// TIA Portal V17 export
// export: Created 2025-06-20T10:18:09.7290963Z, ExportSetting WithDefaults, DisplayName Totally Integrated Automation Portal, DisplayVersion V17 Update 8, DisplayName TIA Portal Openness, DisplayVersion V17 Update 8, DisplayName TIA Portal Version Control Interface, DisplayVersion V17, DisplayName SINAMICS Startdrive Advanced, DisplayVersion V17 SP2, DisplayName SINAMICS Startdrive G110M, G120, G120C, G120D, G120P, G115D, DisplayVersion V17 SP2, DisplayName SINAMICS Startdrive G130, G150, S120, S150, SINAMICS MV, S210, DisplayVersion V17 SP2, DisplayName STEP 7 Professional, DisplayVersion V17 Update 8, DisplayName SINUMERIK ONE STEP 7 Toolbox, DisplayVersion V17 Update 12, DisplayName SINUMERIK ONE PLC Basic Program Plus, DisplayVersion V17 Update 12, DisplayName SINUMERIK 840D sl STEP 7 Toolbox, DisplayVersion V17 Update 12, DisplayName STEP 7 Safety, DisplayVersion V17 Update 6, DisplayName WinCC Advanced, DisplayVersion V17 Update 8
FUNCTION "FC370_NCK_M_CH8_UNIT_03" : Void   // FC370, LAD
TITLE = Channel 1 data
{ S7_Optimized_Access := 'FALSE' }
AUTHOR : ETXETAR
VERSION : 1.0
// stored: AutoNumber false, IsIECCheckEnabled false, SetENOAutomatically false, UDAEnableTagReadback false
BEGIN

REGION Network 1: ACKNOWLEDGE M704-FIXTURE 4 VERIFY PART AND TOOL IS CLAMPED DURING MACHINING (WHEN TRUE DO). TOGGLED / ACKNOWLEDGE M46-VERIFY FIXTURE 1 PART AND TOOL IS CLAMPED DURING
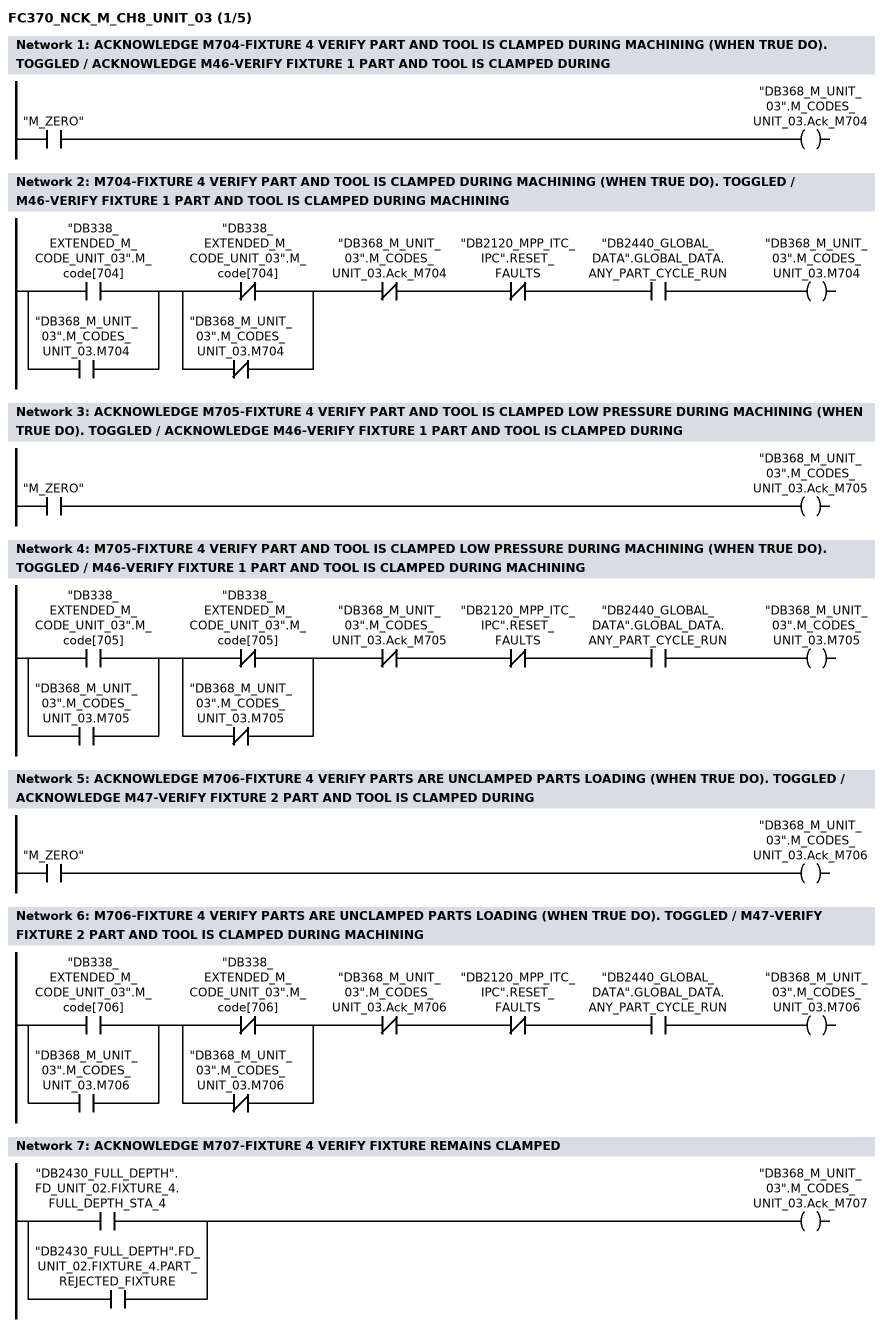
   RUNG wire#powerrail
      Contact( "M_ZERO" )
      Coil( "DB368_M_UNIT_03".M_CODES_UNIT_03.Ack_M704 )
   END_RUNG
   // the same network as SCL:
   "DB368_M_UNIT_03".M_CODES_UNIT_03.Ack_M704 := "M_ZERO";
END_REGION

REGION Network 2: M704-FIXTURE 4 VERIFY PART AND TOOL IS CLAMPED DURING MACHINING (WHEN TRUE DO). TOGGLED / M46-VERIFY FIXTURE 1 PART AND TOOL IS CLAMPED DURING MACHINING
   RUNG wire#powerrail
      Contact( "DB338_EXTENDED_M_CODE_UNIT_03".M_code[704] )
      wire#w1
      I_Contact( "DB338_EXTENDED_M_CODE_UNIT_03".M_code[704] )
      wire#w2
      I_Contact( "DB368_M_UNIT_03".M_CODES_UNIT_03.Ack_M704 )
      I_Contact( "DB2120_MPP_ITC_IPC".RESET_FAULTS )
      Contact( "DB2440_GLOBAL_DATA".GLOBAL_DATA.ANY_PART_CYCLE_RUN )
      Coil( "DB368_M_UNIT_03".M_CODES_UNIT_03.M704 )
   END_RUNG
   RUNG wire#powerrail
      Contact( "DB368_M_UNIT_03".M_CODES_UNIT_03.M704 )
   END_RUNG wire#w1
   RUNG wire#w1
      I_Contact( "DB368_M_UNIT_03".M_CODES_UNIT_03.M704 )
   END_RUNG wire#w2
   // the same network as SCL:
   "DB368_M_UNIT_03".M_CODES_UNIT_03.M704 := ("DB338_EXTENDED_M_CODE_UNIT_03".M_code[704] OR "DB368_M_UNIT_03".M_CODES_UNIT_03.M704) AND (NOT "DB338_EXTENDED_M_CODE_UNIT_03".M_code[704] OR NOT "DB368_M_UNIT_03".M_CODES_UNIT_03.M704) AND NOT "DB368_M_UNIT_03".M_CODES_UNIT_03.Ack_M704 AND NOT "DB2120_MPP_ITC_IPC".RESET_FAULTS AND "DB2440_GLOBAL_DATA".GLOBAL_DATA.ANY_PART_CYCLE_RUN;
END_REGION

REGION Network 3: ACKNOWLEDGE M705-FIXTURE 4 VERIFY PART AND TOOL IS CLAMPED LOW PRESSURE DURING MACHINING (WHEN TRUE DO). TOGGLED / ACKNOWLEDGE M46-VERIFY FIXTURE 1 PART AND TOOL IS CLAMPED DURING
   RUNG wire#powerrail
      Contact( "M_ZERO" )
      Coil( "DB368_M_UNIT_03".M_CODES_UNIT_03.Ack_M705 )
   END_RUNG
   // the same network as SCL:
   "DB368_M_UNIT_03".M_CODES_UNIT_03.Ack_M705 := "M_ZERO";
END_REGION

REGION Network 4: M705-FIXTURE 4 VERIFY PART AND TOOL IS CLAMPED LOW PRESSURE DURING MACHINING (WHEN TRUE DO). TOGGLED / M46-VERIFY FIXTURE 1 PART AND TOOL IS CLAMPED DURING MACHINING
   RUNG wire#powerrail
      Contact( "DB338_EXTENDED_M_CODE_UNIT_03".M_code[705] )
      wire#w1
      I_Contact( "DB338_EXTENDED_M_CODE_UNIT_03".M_code[705] )
      wire#w2
      I_Contact( "DB368_M_UNIT_03".M_CODES_UNIT_03.Ack_M705 )
      I_Contact( "DB2120_MPP_ITC_IPC".RESET_FAULTS )
      Contact( "DB2440_GLOBAL_DATA".GLOBAL_DATA.ANY_PART_CYCLE_RUN )
      Coil( "DB368_M_UNIT_03".M_CODES_UNIT_03.M705 )
   END_RUNG
   RUNG wire#powerrail
      Contact( "DB368_M_UNIT_03".M_CODES_UNIT_03.M705 )
   END_RUNG wire#w1
   RUNG wire#w1
      I_Contact( "DB368_M_UNIT_03".M_CODES_UNIT_03.M705 )
   END_RUNG wire#w2
   // the same network as SCL:
   "DB368_M_UNIT_03".M_CODES_UNIT_03.M705 := ("DB338_EXTENDED_M_CODE_UNIT_03".M_code[705] OR "DB368_M_UNIT_03".M_CODES_UNIT_03.M705) AND (NOT "DB338_EXTENDED_M_CODE_UNIT_03".M_code[705] OR NOT "DB368_M_UNIT_03".M_CODES_UNIT_03.M705) AND NOT "DB368_M_UNIT_03".M_CODES_UNIT_03.Ack_M705 AND NOT "DB2120_MPP_ITC_IPC".RESET_FAULTS AND "DB2440_GLOBAL_DATA".GLOBAL_DATA.ANY_PART_CYCLE_RUN;
END_REGION

REGION Network 5: ACKNOWLEDGE M706-FIXTURE 4 VERIFY PARTS ARE UNCLAMPED PARTS LOADING (WHEN TRUE DO). TOGGLED / ACKNOWLEDGE M47-VERIFY FIXTURE 2 PART AND TOOL IS CLAMPED DURING
   RUNG wire#powerrail
      Contact( "M_ZERO" )
      Coil( "DB368_M_UNIT_03".M_CODES_UNIT_03.Ack_M706 )
   END_RUNG
   // the same network as SCL:
   "DB368_M_UNIT_03".M_CODES_UNIT_03.Ack_M706 := "M_ZERO";
END_REGION

REGION Network 6: M706-FIXTURE 4 VERIFY PARTS ARE UNCLAMPED PARTS LOADING (WHEN TRUE DO). TOGGLED / M47-VERIFY FIXTURE 2 PART AND TOOL IS CLAMPED DURING MACHINING
   RUNG wire#powerrail
      Contact( "DB338_EXTENDED_M_CODE_UNIT_03".M_code[706] )
      wire#w1
      I_Contact( "DB338_EXTENDED_M_CODE_UNIT_03".M_code[706] )
      wire#w2
      I_Contact( "DB368_M_UNIT_03".M_CODES_UNIT_03.Ack_M706 )
      I_Contact( "DB2120_MPP_ITC_IPC".RESET_FAULTS )
      Contact( "DB2440_GLOBAL_DATA".GLOBAL_DATA.ANY_PART_CYCLE_RUN )
      Coil( "DB368_M_UNIT_03".M_CODES_UNIT_03.M706 )
   END_RUNG
   RUNG wire#powerrail
      Contact( "DB368_M_UNIT_03".M_CODES_UNIT_03.M706 )
   END_RUNG wire#w1
   RUNG wire#w1
      I_Contact( "DB368_M_UNIT_03".M_CODES_UNIT_03.M706 )
   END_RUNG wire#w2
   // the same network as SCL:
   "DB368_M_UNIT_03".M_CODES_UNIT_03.M706 := ("DB338_EXTENDED_M_CODE_UNIT_03".M_code[706] OR "DB368_M_UNIT_03".M_CODES_UNIT_03.M706) AND (NOT "DB338_EXTENDED_M_CODE_UNIT_03".M_code[706] OR NOT "DB368_M_UNIT_03".M_CODES_UNIT_03.M706) AND NOT "DB368_M_UNIT_03".M_CODES_UNIT_03.Ack_M706 AND NOT "DB2120_MPP_ITC_IPC".RESET_FAULTS AND "DB2440_GLOBAL_DATA".GLOBAL_DATA.ANY_PART_CYCLE_RUN;
END_REGION

REGION Network 7: ACKNOWLEDGE M707-FIXTURE 4 VERIFY FIXTURE REMAINS CLAMPED
   RUNG wire#powerrail
      Contact( "DB2430_FULL_DEPTH".FD_UNIT_02.FIXTURE_4.FULL_DEPTH_STA_4 )
      wire#w1
      Coil( "DB368_M_UNIT_03".M_CODES_UNIT_03.Ack_M707 )
   END_RUNG
   RUNG wire#powerrail
      Contact( "DB2430_FULL_DEPTH".FD_UNIT_02.FIXTURE_4.PART_REJECTED_FIXTURE )
   END_RUNG wire#w1
   // the same network as SCL:
   "DB368_M_UNIT_03".M_CODES_UNIT_03.Ack_M707 := "DB2430_FULL_DEPTH".FD_UNIT_02.FIXTURE_4.FULL_DEPTH_STA_4 OR "DB2430_FULL_DEPTH".FD_UNIT_02.FIXTURE_4.PART_REJECTED_FIXTURE;
END_REGION

REGION Network 8: M707-FIXTURE 4 VERIFY FIXTURE REMAINS CLAMPED
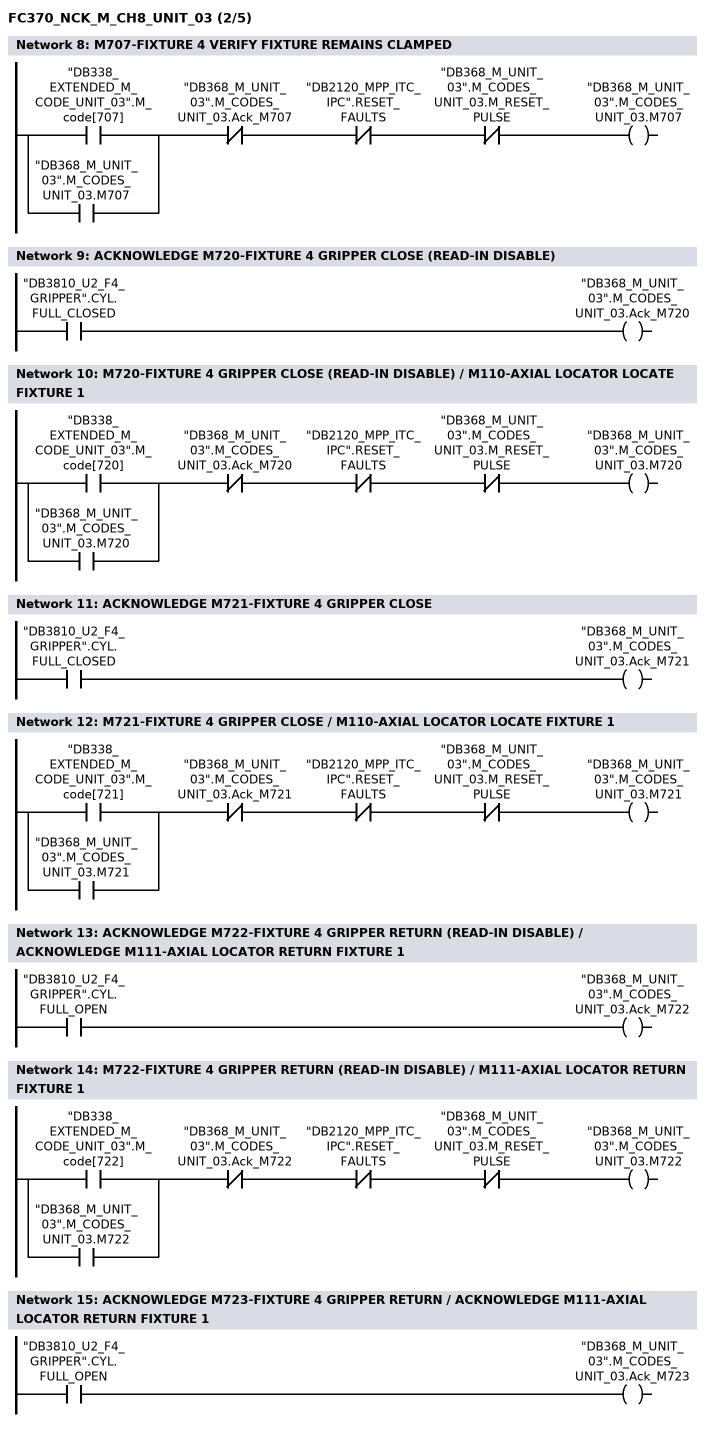
   RUNG wire#powerrail
      Contact( "DB338_EXTENDED_M_CODE_UNIT_03".M_code[707] )
      wire#w1
      I_Contact( "DB368_M_UNIT_03".M_CODES_UNIT_03.Ack_M707 )
      I_Contact( "DB2120_MPP_ITC_IPC".RESET_FAULTS )
      I_Contact( "DB368_M_UNIT_03".M_CODES_UNIT_03.M_RESET_PULSE )
      Coil( "DB368_M_UNIT_03".M_CODES_UNIT_03.M707 )
   END_RUNG
   RUNG wire#powerrail
      Contact( "DB368_M_UNIT_03".M_CODES_UNIT_03.M707 )
   END_RUNG wire#w1
   // the same network as SCL:
   "DB368_M_UNIT_03".M_CODES_UNIT_03.M707 := ("DB338_EXTENDED_M_CODE_UNIT_03".M_code[707] OR "DB368_M_UNIT_03".M_CODES_UNIT_03.M707) AND NOT "DB368_M_UNIT_03".M_CODES_UNIT_03.Ack_M707 AND NOT "DB2120_MPP_ITC_IPC".RESET_FAULTS AND NOT "DB368_M_UNIT_03".M_CODES_UNIT_03.M_RESET_PULSE;
END_REGION

REGION Network 9: ACKNOWLEDGE M720-FIXTURE 4 GRIPPER CLOSE (READ-IN DISABLE)
   RUNG wire#powerrail
      Contact( "DB3810_U2_F4_GRIPPER".CYL.FULL_CLOSED )
      Coil( "DB368_M_UNIT_03".M_CODES_UNIT_03.Ack_M720 )
   END_RUNG
   // the same network as SCL:
   "DB368_M_UNIT_03".M_CODES_UNIT_03.Ack_M720 := "DB3810_U2_F4_GRIPPER".CYL.FULL_CLOSED;
END_REGION

REGION Network 10: M720-FIXTURE 4 GRIPPER CLOSE (READ-IN DISABLE) / M110-AXIAL LOCATOR LOCATE FIXTURE 1
   RUNG wire#powerrail
      Contact( "DB338_EXTENDED_M_CODE_UNIT_03".M_code[720] )
      wire#w1
      I_Contact( "DB368_M_UNIT_03".M_CODES_UNIT_03.Ack_M720 )
      I_Contact( "DB2120_MPP_ITC_IPC".RESET_FAULTS )
      I_Contact( "DB368_M_UNIT_03".M_CODES_UNIT_03.M_RESET_PULSE )
      Coil( "DB368_M_UNIT_03".M_CODES_UNIT_03.M720 )
   END_RUNG
   RUNG wire#powerrail
      Contact( "DB368_M_UNIT_03".M_CODES_UNIT_03.M720 )
   END_RUNG wire#w1
   // the same network as SCL:
   "DB368_M_UNIT_03".M_CODES_UNIT_03.M720 := ("DB338_EXTENDED_M_CODE_UNIT_03".M_code[720] OR "DB368_M_UNIT_03".M_CODES_UNIT_03.M720) AND NOT "DB368_M_UNIT_03".M_CODES_UNIT_03.Ack_M720 AND NOT "DB2120_MPP_ITC_IPC".RESET_FAULTS AND NOT "DB368_M_UNIT_03".M_CODES_UNIT_03.M_RESET_PULSE;
END_REGION

REGION Network 11: ACKNOWLEDGE M721-FIXTURE 4 GRIPPER CLOSE
   RUNG wire#powerrail
      Contact( "DB3810_U2_F4_GRIPPER".CYL.FULL_CLOSED )
      Coil( "DB368_M_UNIT_03".M_CODES_UNIT_03.Ack_M721 )
   END_RUNG
   // the same network as SCL:
   "DB368_M_UNIT_03".M_CODES_UNIT_03.Ack_M721 := "DB3810_U2_F4_GRIPPER".CYL.FULL_CLOSED;
END_REGION

REGION Network 12: M721-FIXTURE 4 GRIPPER CLOSE / M110-AXIAL LOCATOR LOCATE FIXTURE 1
   RUNG wire#powerrail
      Contact( "DB338_EXTENDED_M_CODE_UNIT_03".M_code[721] )
      wire#w1
      I_Contact( "DB368_M_UNIT_03".M_CODES_UNIT_03.Ack_M721 )
      I_Contact( "DB2120_MPP_ITC_IPC".RESET_FAULTS )
      I_Contact( "DB368_M_UNIT_03".M_CODES_UNIT_03.M_RESET_PULSE )
      Coil( "DB368_M_UNIT_03".M_CODES_UNIT_03.M721 )
   END_RUNG
   RUNG wire#powerrail
      Contact( "DB368_M_UNIT_03".M_CODES_UNIT_03.M721 )
   END_RUNG wire#w1
   // the same network as SCL:
   "DB368_M_UNIT_03".M_CODES_UNIT_03.M721 := ("DB338_EXTENDED_M_CODE_UNIT_03".M_code[721] OR "DB368_M_UNIT_03".M_CODES_UNIT_03.M721) AND NOT "DB368_M_UNIT_03".M_CODES_UNIT_03.Ack_M721 AND NOT "DB2120_MPP_ITC_IPC".RESET_FAULTS AND NOT "DB368_M_UNIT_03".M_CODES_UNIT_03.M_RESET_PULSE;
END_REGION

REGION Network 13: ACKNOWLEDGE M722-FIXTURE 4 GRIPPER RETURN (READ-IN DISABLE) / ACKNOWLEDGE M111-AXIAL LOCATOR RETURN FIXTURE 1
   RUNG wire#powerrail
      Contact( "DB3810_U2_F4_GRIPPER".CYL.FULL_OPEN )
      Coil( "DB368_M_UNIT_03".M_CODES_UNIT_03.Ack_M722 )
   END_RUNG
   // the same network as SCL:
   "DB368_M_UNIT_03".M_CODES_UNIT_03.Ack_M722 := "DB3810_U2_F4_GRIPPER".CYL.FULL_OPEN;
END_REGION

REGION Network 14: M722-FIXTURE 4 GRIPPER RETURN (READ-IN DISABLE) / M111-AXIAL LOCATOR RETURN FIXTURE 1
   RUNG wire#powerrail
      Contact( "DB338_EXTENDED_M_CODE_UNIT_03".M_code[722] )
      wire#w1
      I_Contact( "DB368_M_UNIT_03".M_CODES_UNIT_03.Ack_M722 )
      I_Contact( "DB2120_MPP_ITC_IPC".RESET_FAULTS )
      I_Contact( "DB368_M_UNIT_03".M_CODES_UNIT_03.M_RESET_PULSE )
      Coil( "DB368_M_UNIT_03".M_CODES_UNIT_03.M722 )
   END_RUNG
   RUNG wire#powerrail
      Contact( "DB368_M_UNIT_03".M_CODES_UNIT_03.M722 )
   END_RUNG wire#w1
   // the same network as SCL:
   "DB368_M_UNIT_03".M_CODES_UNIT_03.M722 := ("DB338_EXTENDED_M_CODE_UNIT_03".M_code[722] OR "DB368_M_UNIT_03".M_CODES_UNIT_03.M722) AND NOT "DB368_M_UNIT_03".M_CODES_UNIT_03.Ack_M722 AND NOT "DB2120_MPP_ITC_IPC".RESET_FAULTS AND NOT "DB368_M_UNIT_03".M_CODES_UNIT_03.M_RESET_PULSE;
END_REGION

REGION Network 15: ACKNOWLEDGE M723-FIXTURE 4 GRIPPER RETURN / ACKNOWLEDGE M111-AXIAL LOCATOR RETURN FIXTURE 1
   RUNG wire#powerrail
      Contact( "DB3810_U2_F4_GRIPPER".CYL.FULL_OPEN )
      Coil( "DB368_M_UNIT_03".M_CODES_UNIT_03.Ack_M723 )
   END_RUNG
   // the same network as SCL:
   "DB368_M_UNIT_03".M_CODES_UNIT_03.Ack_M723 := "DB3810_U2_F4_GRIPPER".CYL.FULL_OPEN;
END_REGION

REGION Network 16: M723-FIXTURE 4 GRIPPER RETURN / M111-AXIAL LOCATOR RETURN FIXTURE 1
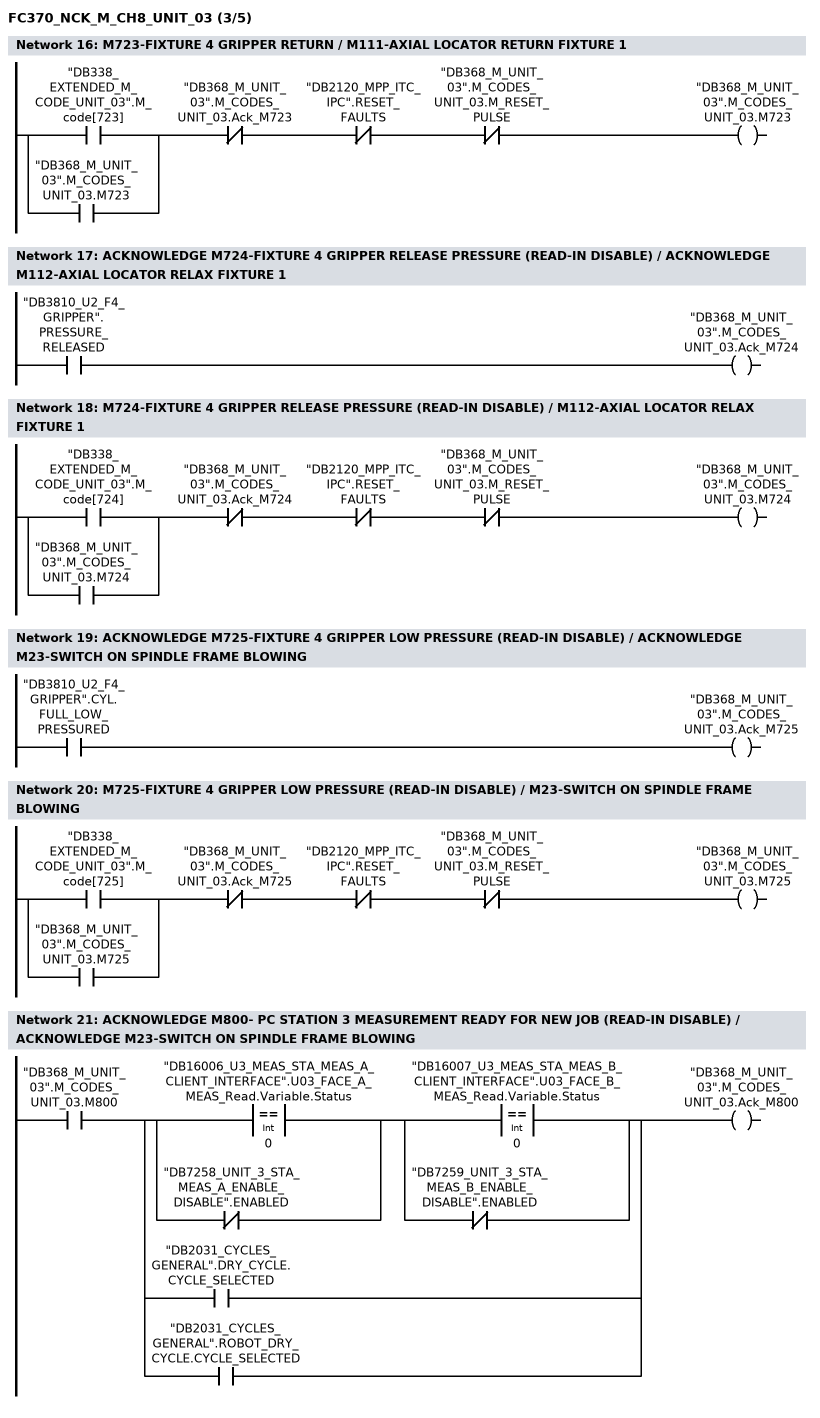
   RUNG wire#powerrail
      Contact( "DB338_EXTENDED_M_CODE_UNIT_03".M_code[723] )
      wire#w1
      I_Contact( "DB368_M_UNIT_03".M_CODES_UNIT_03.Ack_M723 )
      I_Contact( "DB2120_MPP_ITC_IPC".RESET_FAULTS )
      I_Contact( "DB368_M_UNIT_03".M_CODES_UNIT_03.M_RESET_PULSE )
      Coil( "DB368_M_UNIT_03".M_CODES_UNIT_03.M723 )
   END_RUNG
   RUNG wire#powerrail
      Contact( "DB368_M_UNIT_03".M_CODES_UNIT_03.M723 )
   END_RUNG wire#w1
   // the same network as SCL:
   "DB368_M_UNIT_03".M_CODES_UNIT_03.M723 := ("DB338_EXTENDED_M_CODE_UNIT_03".M_code[723] OR "DB368_M_UNIT_03".M_CODES_UNIT_03.M723) AND NOT "DB368_M_UNIT_03".M_CODES_UNIT_03.Ack_M723 AND NOT "DB2120_MPP_ITC_IPC".RESET_FAULTS AND NOT "DB368_M_UNIT_03".M_CODES_UNIT_03.M_RESET_PULSE;
END_REGION

REGION Network 17: ACKNOWLEDGE M724-FIXTURE 4 GRIPPER RELEASE PRESSURE (READ-IN DISABLE) / ACKNOWLEDGE M112-AXIAL LOCATOR RELAX FIXTURE 1
   RUNG wire#powerrail
      Contact( "DB3810_U2_F4_GRIPPER".PRESSURE_RELEASED )
      Coil( "DB368_M_UNIT_03".M_CODES_UNIT_03.Ack_M724 )
   END_RUNG
   // the same network as SCL:
   "DB368_M_UNIT_03".M_CODES_UNIT_03.Ack_M724 := "DB3810_U2_F4_GRIPPER".PRESSURE_RELEASED;
END_REGION

REGION Network 18: M724-FIXTURE 4 GRIPPER RELEASE PRESSURE (READ-IN DISABLE) / M112-AXIAL LOCATOR RELAX FIXTURE 1
   RUNG wire#powerrail
      Contact( "DB338_EXTENDED_M_CODE_UNIT_03".M_code[724] )
      wire#w1
      I_Contact( "DB368_M_UNIT_03".M_CODES_UNIT_03.Ack_M724 )
      I_Contact( "DB2120_MPP_ITC_IPC".RESET_FAULTS )
      I_Contact( "DB368_M_UNIT_03".M_CODES_UNIT_03.M_RESET_PULSE )
      Coil( "DB368_M_UNIT_03".M_CODES_UNIT_03.M724 )
   END_RUNG
   RUNG wire#powerrail
      Contact( "DB368_M_UNIT_03".M_CODES_UNIT_03.M724 )
   END_RUNG wire#w1
   // the same network as SCL:
   "DB368_M_UNIT_03".M_CODES_UNIT_03.M724 := ("DB338_EXTENDED_M_CODE_UNIT_03".M_code[724] OR "DB368_M_UNIT_03".M_CODES_UNIT_03.M724) AND NOT "DB368_M_UNIT_03".M_CODES_UNIT_03.Ack_M724 AND NOT "DB2120_MPP_ITC_IPC".RESET_FAULTS AND NOT "DB368_M_UNIT_03".M_CODES_UNIT_03.M_RESET_PULSE;
END_REGION

REGION Network 19: ACKNOWLEDGE M725-FIXTURE 4 GRIPPER LOW PRESSURE (READ-IN DISABLE) / ACKNOWLEDGE M23-SWITCH ON SPINDLE FRAME BLOWING
   RUNG wire#powerrail
      Contact( "DB3810_U2_F4_GRIPPER".CYL.FULL_LOW_PRESSURED )
      Coil( "DB368_M_UNIT_03".M_CODES_UNIT_03.Ack_M725 )
   END_RUNG
   // the same network as SCL:
   "DB368_M_UNIT_03".M_CODES_UNIT_03.Ack_M725 := "DB3810_U2_F4_GRIPPER".CYL.FULL_LOW_PRESSURED;
END_REGION

REGION Network 20: M725-FIXTURE 4 GRIPPER LOW PRESSURE (READ-IN DISABLE) / M23-SWITCH ON SPINDLE FRAME BLOWING
   RUNG wire#powerrail
      Contact( "DB338_EXTENDED_M_CODE_UNIT_03".M_code[725] )
      wire#w1
      I_Contact( "DB368_M_UNIT_03".M_CODES_UNIT_03.Ack_M725 )
      I_Contact( "DB2120_MPP_ITC_IPC".RESET_FAULTS )
      I_Contact( "DB368_M_UNIT_03".M_CODES_UNIT_03.M_RESET_PULSE )
      Coil( "DB368_M_UNIT_03".M_CODES_UNIT_03.M725 )
   END_RUNG
   RUNG wire#powerrail
      Contact( "DB368_M_UNIT_03".M_CODES_UNIT_03.M725 )
   END_RUNG wire#w1
   // the same network as SCL:
   "DB368_M_UNIT_03".M_CODES_UNIT_03.M725 := ("DB338_EXTENDED_M_CODE_UNIT_03".M_code[725] OR "DB368_M_UNIT_03".M_CODES_UNIT_03.M725) AND NOT "DB368_M_UNIT_03".M_CODES_UNIT_03.Ack_M725 AND NOT "DB2120_MPP_ITC_IPC".RESET_FAULTS AND NOT "DB368_M_UNIT_03".M_CODES_UNIT_03.M_RESET_PULSE;
END_REGION

REGION Network 21: ACKNOWLEDGE M800- PC STATION 3 MEASUREMENT READY FOR NEW JOB (READ-IN DISABLE) / ACKNOWLEDGE M23-SWITCH ON SPINDLE FRAME BLOWING
   RUNG wire#powerrail
      Contact( "DB368_M_UNIT_03".M_CODES_UNIT_03.M800 )
      wire#w1
      { S7_Templates := "SrcType := Int" } EQ_Contact(in1 := "DB16006_U3_MEAS_STA_MEAS_A_CLIENT_INTERFACE".U03_FACE_A_MEAS_Read.Variable.Status, in2 := 0)
      wire#w2
      { S7_Templates := "SrcType := Int" } EQ_Contact(in1 := "DB16007_U3_MEAS_STA_MEAS_B_CLIENT_INTERFACE".U03_FACE_B_MEAS_Read.Variable.Status, in2 := 0)
      wire#w3
      Coil( "DB368_M_UNIT_03".M_CODES_UNIT_03.Ack_M800 )
   END_RUNG
   RUNG wire#w1
      I_Contact( "DB7258_UNIT_3_STA_MEAS_A_ENABLE_DISABLE".ENABLED )
   END_RUNG wire#w2
   RUNG wire#w2
      I_Contact( "DB7259_UNIT_3_STA_MEAS_B_ENABLE_DISABLE".ENABLED )
   END_RUNG wire#w3
   RUNG wire#w1
      Contact( "DB2031_CYCLES_GENERAL".DRY_CYCLE.CYCLE_SELECTED )
   END_RUNG wire#w3
   RUNG wire#w1
      Contact( "DB2031_CYCLES_GENERAL".ROBOT_DRY_CYCLE.CYCLE_SELECTED )
   END_RUNG wire#w3
   // the same network as SCL:
   "DB368_M_UNIT_03".M_CODES_UNIT_03.Ack_M800 := "DB368_M_UNIT_03".M_CODES_UNIT_03.M800 AND (((("DB16006_U3_MEAS_STA_MEAS_A_CLIENT_INTERFACE".U03_FACE_A_MEAS_Read.Variable.Status = 0) OR NOT "DB7258_UNIT_3_STA_MEAS_A_ENABLE_DISABLE".ENABLED) AND (("DB16007_U3_MEAS_STA_MEAS_B_CLIENT_INTERFACE".U03_FACE_B_MEAS_Read.Variable.Status = 0) OR NOT "DB7259_UNIT_3_STA_MEAS_B_ENABLE_DISABLE".ENABLED)) OR "DB2031_CYCLES_GENERAL".DRY_CYCLE.CYCLE_SELECTED OR "DB2031_CYCLES_GENERAL".ROBOT_DRY_CYCLE.CYCLE_SELECTED);
END_REGION

REGION Network 22: M800- PC STATION 3 MEASUREMENT READY FOR NEW JOB (READ-IN DISABLE) / M23-SWITCH ON SPINDLE FRAME BLOWING
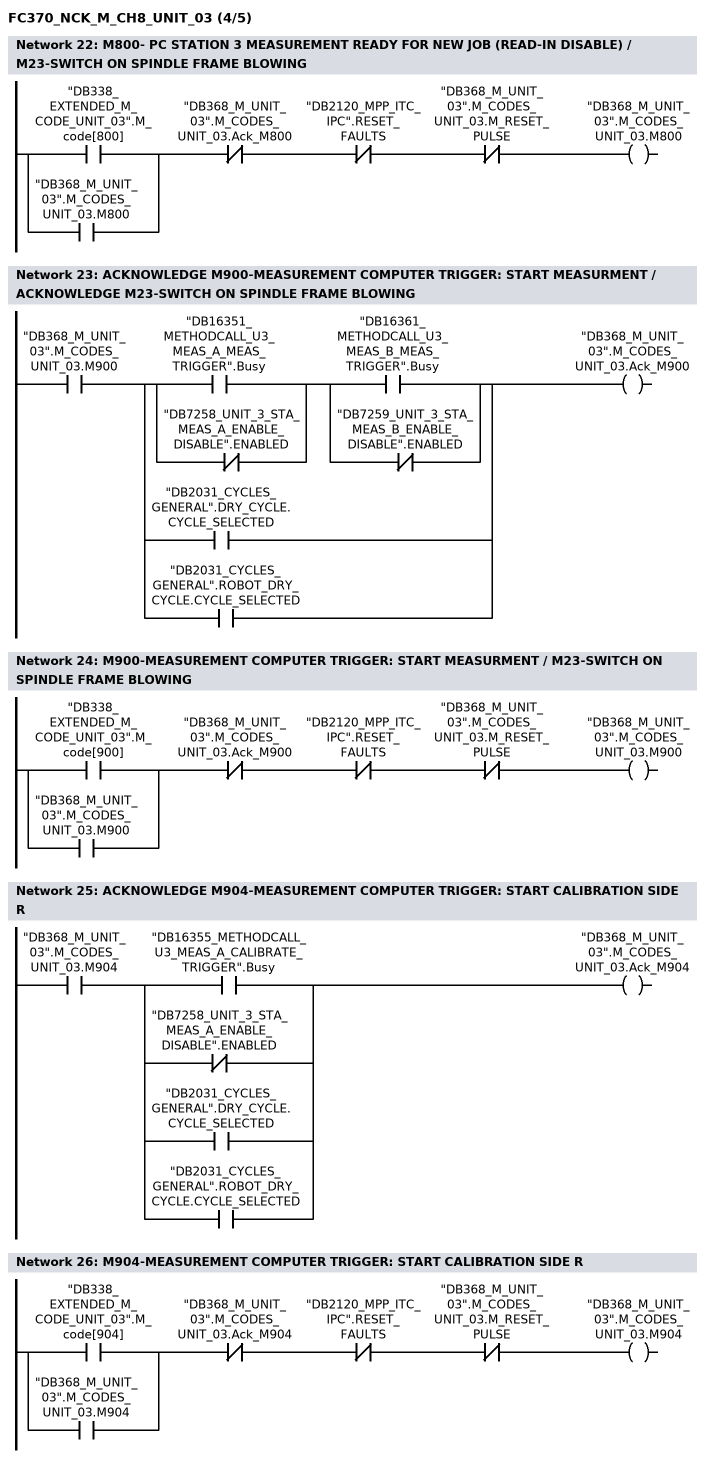
   RUNG wire#powerrail
      Contact( "DB338_EXTENDED_M_CODE_UNIT_03".M_code[800] )
      wire#w1
      I_Contact( "DB368_M_UNIT_03".M_CODES_UNIT_03.Ack_M800 )
      I_Contact( "DB2120_MPP_ITC_IPC".RESET_FAULTS )
      I_Contact( "DB368_M_UNIT_03".M_CODES_UNIT_03.M_RESET_PULSE )
      Coil( "DB368_M_UNIT_03".M_CODES_UNIT_03.M800 )
   END_RUNG
   RUNG wire#powerrail
      Contact( "DB368_M_UNIT_03".M_CODES_UNIT_03.M800 )
   END_RUNG wire#w1
   // the same network as SCL:
   "DB368_M_UNIT_03".M_CODES_UNIT_03.M800 := ("DB338_EXTENDED_M_CODE_UNIT_03".M_code[800] OR "DB368_M_UNIT_03".M_CODES_UNIT_03.M800) AND NOT "DB368_M_UNIT_03".M_CODES_UNIT_03.Ack_M800 AND NOT "DB2120_MPP_ITC_IPC".RESET_FAULTS AND NOT "DB368_M_UNIT_03".M_CODES_UNIT_03.M_RESET_PULSE;
END_REGION

REGION Network 23: ACKNOWLEDGE M900-MEASUREMENT COMPUTER TRIGGER: START MEASURMENT / ACKNOWLEDGE M23-SWITCH ON SPINDLE FRAME BLOWING
   RUNG wire#powerrail
      Contact( "DB368_M_UNIT_03".M_CODES_UNIT_03.M900 )
      wire#w1
      Contact( "DB16351_METHODCALL_U3_MEAS_A_MEAS_TRIGGER".Busy )
      wire#w2
      Contact( "DB16361_METHODCALL_U3_MEAS_B_MEAS_TRIGGER".Busy )
      wire#w3
      Coil( "DB368_M_UNIT_03".M_CODES_UNIT_03.Ack_M900 )
   END_RUNG
   RUNG wire#w1
      I_Contact( "DB7258_UNIT_3_STA_MEAS_A_ENABLE_DISABLE".ENABLED )
   END_RUNG wire#w2
   RUNG wire#w2
      I_Contact( "DB7259_UNIT_3_STA_MEAS_B_ENABLE_DISABLE".ENABLED )
   END_RUNG wire#w3
   RUNG wire#w1
      Contact( "DB2031_CYCLES_GENERAL".DRY_CYCLE.CYCLE_SELECTED )
   END_RUNG wire#w3
   RUNG wire#w1
      Contact( "DB2031_CYCLES_GENERAL".ROBOT_DRY_CYCLE.CYCLE_SELECTED )
   END_RUNG wire#w3
   // the same network as SCL:
   "DB368_M_UNIT_03".M_CODES_UNIT_03.Ack_M900 := "DB368_M_UNIT_03".M_CODES_UNIT_03.M900 AND ((("DB16351_METHODCALL_U3_MEAS_A_MEAS_TRIGGER".Busy OR NOT "DB7258_UNIT_3_STA_MEAS_A_ENABLE_DISABLE".ENABLED) AND ("DB16361_METHODCALL_U3_MEAS_B_MEAS_TRIGGER".Busy OR NOT "DB7259_UNIT_3_STA_MEAS_B_ENABLE_DISABLE".ENABLED)) OR "DB2031_CYCLES_GENERAL".DRY_CYCLE.CYCLE_SELECTED OR "DB2031_CYCLES_GENERAL".ROBOT_DRY_CYCLE.CYCLE_SELECTED);
END_REGION

REGION Network 24: M900-MEASUREMENT COMPUTER TRIGGER: START MEASURMENT / M23-SWITCH ON SPINDLE FRAME BLOWING
   RUNG wire#powerrail
      Contact( "DB338_EXTENDED_M_CODE_UNIT_03".M_code[900] )
      wire#w1
      I_Contact( "DB368_M_UNIT_03".M_CODES_UNIT_03.Ack_M900 )
      I_Contact( "DB2120_MPP_ITC_IPC".RESET_FAULTS )
      I_Contact( "DB368_M_UNIT_03".M_CODES_UNIT_03.M_RESET_PULSE )
      Coil( "DB368_M_UNIT_03".M_CODES_UNIT_03.M900 )
   END_RUNG
   RUNG wire#powerrail
      Contact( "DB368_M_UNIT_03".M_CODES_UNIT_03.M900 )
   END_RUNG wire#w1
   // the same network as SCL:
   "DB368_M_UNIT_03".M_CODES_UNIT_03.M900 := ("DB338_EXTENDED_M_CODE_UNIT_03".M_code[900] OR "DB368_M_UNIT_03".M_CODES_UNIT_03.M900) AND NOT "DB368_M_UNIT_03".M_CODES_UNIT_03.Ack_M900 AND NOT "DB2120_MPP_ITC_IPC".RESET_FAULTS AND NOT "DB368_M_UNIT_03".M_CODES_UNIT_03.M_RESET_PULSE;
END_REGION

REGION Network 25: ACKNOWLEDGE M904-MEASUREMENT COMPUTER TRIGGER: START CALIBRATION SIDE R
   RUNG wire#powerrail
      Contact( "DB368_M_UNIT_03".M_CODES_UNIT_03.M904 )
      wire#w1
      Contact( "DB16355_METHODCALL_U3_MEAS_A_CALIBRATE_TRIGGER".Busy )
      wire#w2
      Coil( "DB368_M_UNIT_03".M_CODES_UNIT_03.Ack_M904 )
   END_RUNG
   RUNG wire#w1
      I_Contact( "DB7258_UNIT_3_STA_MEAS_A_ENABLE_DISABLE".ENABLED )
   END_RUNG wire#w2
   RUNG wire#w1
      Contact( "DB2031_CYCLES_GENERAL".DRY_CYCLE.CYCLE_SELECTED )
   END_RUNG wire#w2
   RUNG wire#w1
      Contact( "DB2031_CYCLES_GENERAL".ROBOT_DRY_CYCLE.CYCLE_SELECTED )
   END_RUNG wire#w2
   // the same network as SCL:
   "DB368_M_UNIT_03".M_CODES_UNIT_03.Ack_M904 := "DB368_M_UNIT_03".M_CODES_UNIT_03.M904 AND ("DB16355_METHODCALL_U3_MEAS_A_CALIBRATE_TRIGGER".Busy OR NOT "DB7258_UNIT_3_STA_MEAS_A_ENABLE_DISABLE".ENABLED OR "DB2031_CYCLES_GENERAL".DRY_CYCLE.CYCLE_SELECTED OR "DB2031_CYCLES_GENERAL".ROBOT_DRY_CYCLE.CYCLE_SELECTED);
END_REGION

REGION Network 26: M904-MEASUREMENT COMPUTER TRIGGER: START CALIBRATION SIDE R
   RUNG wire#powerrail
      Contact( "DB338_EXTENDED_M_CODE_UNIT_03".M_code[904] )
      wire#w1
      I_Contact( "DB368_M_UNIT_03".M_CODES_UNIT_03.Ack_M904 )
      I_Contact( "DB2120_MPP_ITC_IPC".RESET_FAULTS )
      I_Contact( "DB368_M_UNIT_03".M_CODES_UNIT_03.M_RESET_PULSE )
      Coil( "DB368_M_UNIT_03".M_CODES_UNIT_03.M904 )
   END_RUNG
   RUNG wire#powerrail
      Contact( "DB368_M_UNIT_03".M_CODES_UNIT_03.M904 )
   END_RUNG wire#w1
   // the same network as SCL:
   "DB368_M_UNIT_03".M_CODES_UNIT_03.M904 := ("DB338_EXTENDED_M_CODE_UNIT_03".M_code[904] OR "DB368_M_UNIT_03".M_CODES_UNIT_03.M904) AND NOT "DB368_M_UNIT_03".M_CODES_UNIT_03.Ack_M904 AND NOT "DB2120_MPP_ITC_IPC".RESET_FAULTS AND NOT "DB368_M_UNIT_03".M_CODES_UNIT_03.M_RESET_PULSE;
END_REGION

REGION Network 27: ACKNOWLEDGE M905-MEASUREMENT COMPUTER TRIGGER: START CALIBRATION SIDE N
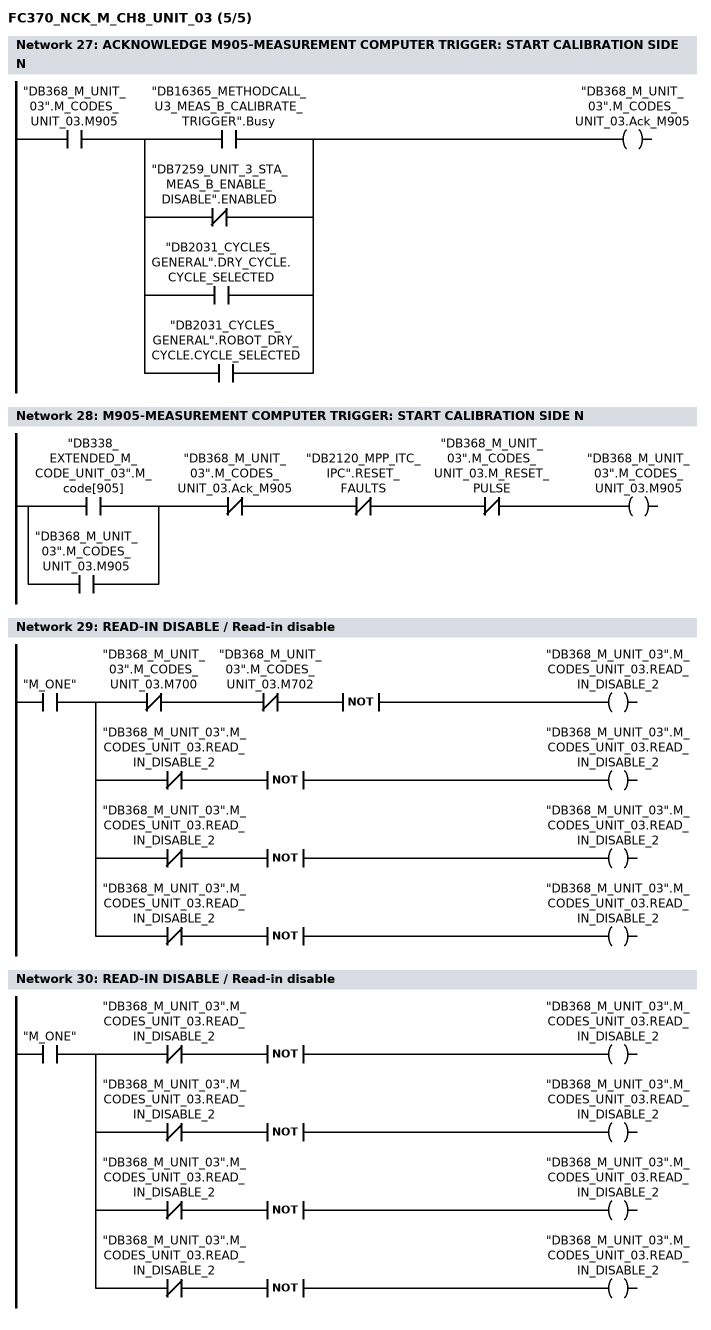
   RUNG wire#powerrail
      Contact( "DB368_M_UNIT_03".M_CODES_UNIT_03.M905 )
      wire#w1
      Contact( "DB16365_METHODCALL_U3_MEAS_B_CALIBRATE_TRIGGER".Busy )
      wire#w2
      Coil( "DB368_M_UNIT_03".M_CODES_UNIT_03.Ack_M905 )
   END_RUNG
   RUNG wire#w1
      I_Contact( "DB7259_UNIT_3_STA_MEAS_B_ENABLE_DISABLE".ENABLED )
   END_RUNG wire#w2
   RUNG wire#w1
      Contact( "DB2031_CYCLES_GENERAL".DRY_CYCLE.CYCLE_SELECTED )
   END_RUNG wire#w2
   RUNG wire#w1
      Contact( "DB2031_CYCLES_GENERAL".ROBOT_DRY_CYCLE.CYCLE_SELECTED )
   END_RUNG wire#w2
   // the same network as SCL:
   "DB368_M_UNIT_03".M_CODES_UNIT_03.Ack_M905 := "DB368_M_UNIT_03".M_CODES_UNIT_03.M905 AND ("DB16365_METHODCALL_U3_MEAS_B_CALIBRATE_TRIGGER".Busy OR NOT "DB7259_UNIT_3_STA_MEAS_B_ENABLE_DISABLE".ENABLED OR "DB2031_CYCLES_GENERAL".DRY_CYCLE.CYCLE_SELECTED OR "DB2031_CYCLES_GENERAL".ROBOT_DRY_CYCLE.CYCLE_SELECTED);
END_REGION

REGION Network 28: M905-MEASUREMENT COMPUTER TRIGGER: START CALIBRATION SIDE N
   RUNG wire#powerrail
      Contact( "DB338_EXTENDED_M_CODE_UNIT_03".M_code[905] )
      wire#w1
      I_Contact( "DB368_M_UNIT_03".M_CODES_UNIT_03.Ack_M905 )
      I_Contact( "DB2120_MPP_ITC_IPC".RESET_FAULTS )
      I_Contact( "DB368_M_UNIT_03".M_CODES_UNIT_03.M_RESET_PULSE )
      Coil( "DB368_M_UNIT_03".M_CODES_UNIT_03.M905 )
   END_RUNG
   RUNG wire#powerrail
      Contact( "DB368_M_UNIT_03".M_CODES_UNIT_03.M905 )
   END_RUNG wire#w1
   // the same network as SCL:
   "DB368_M_UNIT_03".M_CODES_UNIT_03.M905 := ("DB338_EXTENDED_M_CODE_UNIT_03".M_code[905] OR "DB368_M_UNIT_03".M_CODES_UNIT_03.M905) AND NOT "DB368_M_UNIT_03".M_CODES_UNIT_03.Ack_M905 AND NOT "DB2120_MPP_ITC_IPC".RESET_FAULTS AND NOT "DB368_M_UNIT_03".M_CODES_UNIT_03.M_RESET_PULSE;
END_REGION

REGION Network 29: READ-IN DISABLE / Read-in disable
   RUNG wire#powerrail
      Contact( "M_ONE" )
      wire#w1
      I_Contact( "DB368_M_UNIT_03".M_CODES_UNIT_03.M700 )
      I_Contact( "DB368_M_UNIT_03".M_CODES_UNIT_03.M702 )
      Not()
      Coil( "DB368_M_UNIT_03".M_CODES_UNIT_03.READ_IN_DISABLE_2 )
   END_RUNG
   RUNG wire#w1
      I_Contact( "DB368_M_UNIT_03".M_CODES_UNIT_03.READ_IN_DISABLE_2 )
      Not()
      Coil( "DB368_M_UNIT_03".M_CODES_UNIT_03.READ_IN_DISABLE_2 )
   END_RUNG
   RUNG wire#w1
      I_Contact( "DB368_M_UNIT_03".M_CODES_UNIT_03.READ_IN_DISABLE_2 )
      Not()
      Coil( "DB368_M_UNIT_03".M_CODES_UNIT_03.READ_IN_DISABLE_2 )
   END_RUNG
   RUNG wire#w1
      I_Contact( "DB368_M_UNIT_03".M_CODES_UNIT_03.READ_IN_DISABLE_2 )
      Not()
      Coil( "DB368_M_UNIT_03".M_CODES_UNIT_03.READ_IN_DISABLE_2 )
   END_RUNG
   // the same network as SCL:
   "DB368_M_UNIT_03".M_CODES_UNIT_03.READ_IN_DISABLE_2 := NOT ("M_ONE" AND NOT "DB368_M_UNIT_03".M_CODES_UNIT_03.M700 AND NOT "DB368_M_UNIT_03".M_CODES_UNIT_03.M702);
   "DB368_M_UNIT_03".M_CODES_UNIT_03.READ_IN_DISABLE_2 := NOT ("M_ONE" AND NOT "DB368_M_UNIT_03".M_CODES_UNIT_03.READ_IN_DISABLE_2);
   "DB368_M_UNIT_03".M_CODES_UNIT_03.READ_IN_DISABLE_2 := NOT ("M_ONE" AND NOT "DB368_M_UNIT_03".M_CODES_UNIT_03.READ_IN_DISABLE_2);
   "DB368_M_UNIT_03".M_CODES_UNIT_03.READ_IN_DISABLE_2 := NOT ("M_ONE" AND NOT "DB368_M_UNIT_03".M_CODES_UNIT_03.READ_IN_DISABLE_2);
END_REGION

REGION Network 30: READ-IN DISABLE / Read-in disable
   RUNG wire#powerrail
      Contact( "M_ONE" )
      wire#w1
      I_Contact( "DB368_M_UNIT_03".M_CODES_UNIT_03.READ_IN_DISABLE_2 )
      Not()
      Coil( "DB368_M_UNIT_03".M_CODES_UNIT_03.READ_IN_DISABLE_2 )
   END_RUNG
   RUNG wire#w1
      I_Contact( "DB368_M_UNIT_03".M_CODES_UNIT_03.READ_IN_DISABLE_2 )
      Not()
      Coil( "DB368_M_UNIT_03".M_CODES_UNIT_03.READ_IN_DISABLE_2 )
   END_RUNG
   RUNG wire#w1
      I_Contact( "DB368_M_UNIT_03".M_CODES_UNIT_03.READ_IN_DISABLE_2 )
      Not()
      Coil( "DB368_M_UNIT_03".M_CODES_UNIT_03.READ_IN_DISABLE_2 )
   END_RUNG
   RUNG wire#w1
      I_Contact( "DB368_M_UNIT_03".M_CODES_UNIT_03.READ_IN_DISABLE_2 )
      Not()
      Coil( "DB368_M_UNIT_03".M_CODES_UNIT_03.READ_IN_DISABLE_2 )
   END_RUNG
   // the same network as SCL:
   "DB368_M_UNIT_03".M_CODES_UNIT_03.READ_IN_DISABLE_2 := NOT ("M_ONE" AND NOT "DB368_M_UNIT_03".M_CODES_UNIT_03.READ_IN_DISABLE_2);
   "DB368_M_UNIT_03".M_CODES_UNIT_03.READ_IN_DISABLE_2 := NOT ("M_ONE" AND NOT "DB368_M_UNIT_03".M_CODES_UNIT_03.READ_IN_DISABLE_2);
   "DB368_M_UNIT_03".M_CODES_UNIT_03.READ_IN_DISABLE_2 := NOT ("M_ONE" AND NOT "DB368_M_UNIT_03".M_CODES_UNIT_03.READ_IN_DISABLE_2);
   "DB368_M_UNIT_03".M_CODES_UNIT_03.READ_IN_DISABLE_2 := NOT ("M_ONE" AND NOT "DB368_M_UNIT_03".M_CODES_UNIT_03.READ_IN_DISABLE_2);
END_REGION
END_FUNCTION
